// TIA Portal V16 export
// export: Created 2025-05-30T16:30:32.2227796Z, ExportSetting WithDefaults, DisplayName Totally Integrated Automation Portal, DisplayVersion V16, DisplayName TIA Portal Version Control Interface, DisplayVersion V16, DisplayName TIA Portal Openness, DisplayVersion V16, DisplayName STEP 7 Professional, DisplayVersion V16, DisplayName STEP 7 Safety, DisplayVersion V16, DisplayName WinCC Advanced, DisplayVersion V16
DATA_BLOCK "FB_SystemTimeCounter_DB_1"   // DB23
VERSION : 0.1
// stored: AutoNumber true, InstanceOfName FB_SystemTimeCounter, InstanceOfType FB
"FB_SystemTimeCounter"
   // VAR_INPUT
   //    Enable : Bool;
   //    CycleTime : Time;
   // END_VAR
   // VAR_OUTPUT
   //    SystemTime : Time;
   // END_VAR
BEGIN
END_DATA_BLOCK
